// TIA Portal V19 export
VAR_GLOBAL   // PLC tag table "Equipment_Template_DefaultTagTable_8"
   "Tag_49(3)" AT %I30042.0 : Bool;
   "Tag_50(3)" AT %I30042.1 : Bool;
   "Tag_51(3)" AT %I30042.2 : Bool;
   "Tag_52(3)" AT %I30042.3 : Bool;
   "Tag_53(3)" AT %I30042.4 : Bool;
   "Tag_54(3)" AT %I30042.5 : Bool;
   "Tag_55(3)" AT %I30042.6 : Bool;
   "Tag_56(3)" AT %I30042.7 : Bool;
   "Tag_57(3)" AT %I30043.0 : Bool;
   "Tag_58(3)" AT %I30043.1 : Bool;
   "Tag_59(3)" AT %I30043.2 : Bool;
   "Tag_60(3)" AT %I30043.3 : Bool;
   "Tag_61(3)" AT %I30043.4 : Bool;
   "Tag_62(3)" AT %I30043.5 : Bool;
   "Tag_63(3)" AT %I30043.6 : Bool;
   "Tag_64(3)" AT %I30043.7 : Bool;
END_VAR
